ABB RAPID module: 0017732A

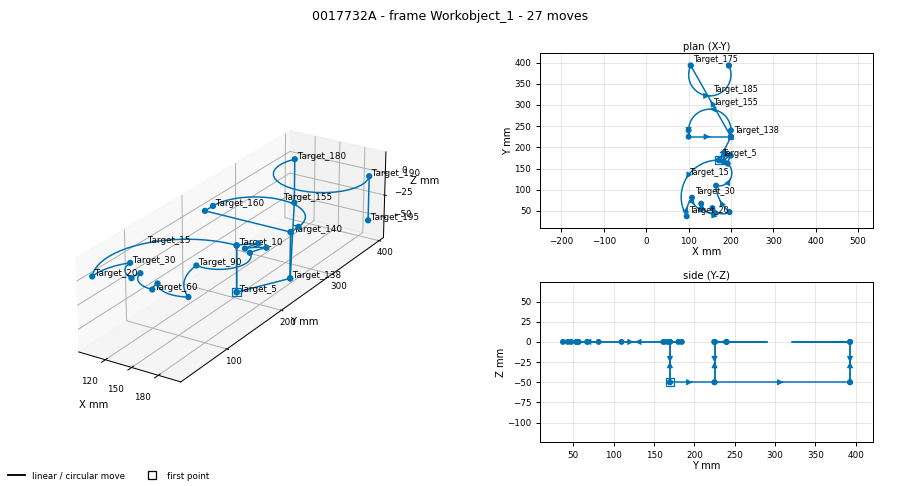
[picture p0: tool path of 0017732A in frame Workobject_1, 27 of 30 moves have a stored position in this frame; points joined in program order, loops and branches not executed]
MODULE Module1
    CONST robtarget Target_M:=[[-410.514648889,1245.713795009,-649.374024814],[0.613768807,0.08026289,-0.406843498,-0.671806585],[0,-1,0,0],[9E+09,9E+09,9E+09,9E+09,9E+09,9E+09]];
    CONST robtarget Target_HH:=[[580.651275023,0,538.588646413],[0.130526193,0,0.991444861,0],[0,0,0,0],[9E+09,9E+09,9E+09,9E+09,9E+09,9E+09]];
    CONST robtarget Target_5:=[[172.146,169.721,-50],[0,0,0,1],[0,0,-1,1],[9E+09,9E+09,9E+09,9E+09,9E+09,9E+09]];
    CONST robtarget Target_10:=[[172.146,169.721,0],[0,0,0,1],[0,0,-1,1],[9E+09,9E+09,9E+09,9E+09,9E+09,9E+09]];
    CONST robtarget Target_15:=[[94.179,126.363,0],[0,0,0,1],[0,0,-1,1],[9E+09,9E+09,9E+09,9E+09,9E+09,9E+09]];
    CONST robtarget Target_20:=[[95.464,37.16,0],[0,0,0,1],[0,0,-1,1],[9E+09,9E+09,9E+09,9E+09,9E+09,9E+09]];
    CONST robtarget Target_25:=[[97.319,60.55,0],[0,0,0,1],[0,0,-1,1],[9E+09,9E+09,9E+09,9E+09,9E+09,9E+09]];
    CONST robtarget Target_30:=[[108.141,81.369,0],[0,0,0,1],[0,0,-1,1],[9E+09,9E+09,9E+09,9E+09,9E+09,9E+09]];
    CONST robtarget Target_35:=[[114.101,64.13,0],[0,0,0,1],[0,0,-1,1],[9E+09,9E+09,9E+09,9E+09,9E+09,9E+09]];
    CONST robtarget Target_40:=[[128.91,53.479,0],[0,0,0,1],[0,0,-1,1],[9E+09,9E+09,9E+09,9E+09,9E+09,9E+09]];
    CONST robtarget Target_45:=[[128.569,60.297,0],[0,0,0,1],[0,0,-1,1],[9E+09,9E+09,9E+09,9E+09,9E+09,9E+09]];
    CONST robtarget Target_50:=[[129.686,67.033,0],[0,0,0,1],[0,0,-1,1],[9E+09,9E+09,9E+09,9E+09,9E+09,9E+09]];
    CONST robtarget Target_55:=[[140.077,49.513,0],[0,0,0,1],[0,0,-1,1],[9E+09,9E+09,9E+09,9E+09,9E+09,9E+09]];
    CONST robtarget Target_60:=[[159.408,43.089,0],[0,0,0,1],[0,0,-1,1],[9E+09,9E+09,9E+09,9E+09,9E+09,9E+09]];
    CONST robtarget Target_65:=[[156.802,49.64,0],[0,0,0,1],[0,0,-1,1],[9E+09,9E+09,9E+09,9E+09,9E+09,9E+09]];
    CONST robtarget Target_70:=[[156.139,56.659,0],[0,0,0,1],[0,0,-1,1],[9E+09,9E+09,9E+09,9E+09,9E+09,9E+09]];
    CONST robtarget Target_75:=[[174.493,43.802,0],[0,0,0,1],[0,0,-1,1],[9E+09,9E+09,9E+09,9E+09,9E+09,9E+09]];
    CONST robtarget Target_80:=[[196.643,47.198,0],[0,0,0,1],[0,0,-1,1],[9E+09,9E+09,9E+09,9E+09,9E+09,9E+09]];
    CONST robtarget Target_85:=[[173.907,75.001,0],[0,0,0,1],[0,0,-1,1],[9E+09,9E+09,9E+09,9E+09,9E+09,9E+09]];
    CONST robtarget Target_90:=[[164.745,109.728,0],[0,0,0,1],[0,0,-1,1],[9E+09,9E+09,9E+09,9E+09,9E+09,9E+09]];
    CONST robtarget Target_95:=[[198.416,125.037,0],[0,0,0,1],[0,0,-1,1],[9E+09,9E+09,9E+09,9E+09,9E+09,9E+09]];
    CONST robtarget Target_100:=[[192.364,161.526,0],[0,0,0,1],[0,0,-1,1],[9E+09,9E+09,9E+09,9E+09,9E+09,9E+09]];
    CONST robtarget Target_105:=[[195.069,171.202,0],[0,0,0,1],[0,0,-1,1],[9E+09,9E+09,9E+09,9E+09,9E+09,9E+09]];
    CONST robtarget Target_110:=[[199.539,180.201,0],[0,0,0,1],[0,0,-1,1],[9E+09,9E+09,9E+09,9E+09,9E+09,9E+09]];
    CONST robtarget Target_115:=[[190.171,175.306,0],[0,0,0,1],[0,0,-1,1],[9E+09,9E+09,9E+09,9E+09,9E+09,9E+09]];
    CONST robtarget Target_120:=[[183.068,167.479,0],[0,0,0,1],[0,0,-1,1],[9E+09,9E+09,9E+09,9E+09,9E+09,9E+09]];
    CONST robtarget Target_125:=[[184.555,176.204,0],[0,0,0,1],[0,0,-1,1],[9E+09,9E+09,9E+09,9E+09,9E+09,9E+09]];
    CONST robtarget Target_130:=[[187.549,184.533,0],[0,0,0,1],[0,0,-1,1],[9E+09,9E+09,9E+09,9E+09,9E+09,9E+09]];
    CONST robtarget Target_135:=[[179.202,177.798,0],[0,0,0,1],[0,0,-1,1],[9E+09,9E+09,9E+09,9E+09,9E+09,9E+09]];
    CONST robtarget Target_138:=[[200,225,-50],[0,0,0,1],[0,-1,0,1],[9E+09,9E+09,9E+09,9E+09,9E+09,9E+09]];
    CONST robtarget Target_140:=[[200,225,0],[0,0,0,1],[0,-1,0,1],[9E+09,9E+09,9E+09,9E+09,9E+09,9E+09]];
    CONST robtarget Target_150:=[[200,240,0],[0,0,0,1],[-1,-1,0,1],[9E+09,9E+09,9E+09,9E+09,9E+09,9E+09]];
    CONST robtarget Target_155:=[[150,290,0],[0,0,0,1],[-1,-1,0,1],[9E+09,9E+09,9E+09,9E+09,9E+09,9E+09]];
    CONST robtarget Target_160:=[[100,240,0],[0,0,0,1],[-1,-1,0,1],[9E+09,9E+09,9E+09,9E+09,9E+09,9E+09]];
    CONST robtarget Target_170:=[[100,225,0],[0,0,0,1],[0,-1,0,1],[9E+09,9E+09,9E+09,9E+09,9E+09,9E+09]];
    CONST robtarget Target_175:=[[105,392.992,-50],[0,0,0,1],[-1,-1,0,1],[9E+09,9E+09,9E+09,9E+09,9E+09,9E+09]];
    CONST robtarget Target_180:=[[105,392.992,0],[0,0,0,1],[-1,-1,0,1],[9E+09,9E+09,9E+09,9E+09,9E+09,9E+09]];
    CONST robtarget Target_185:=[[150,321.197,0],[0,0,0,1],[-1,-1,0,1],[9E+09,9E+09,9E+09,9E+09,9E+09,9E+09]];
    CONST robtarget Target_190:=[[195,392.992,0],[0,0,0,1],[-1,-1,0,1],[9E+09,9E+09,9E+09,9E+09,9E+09,9E+09]];
    CONST robtarget Target_195:=[[195,392.992,-50],[0,0,0,1],[-1,-1,0,1],[9E+09,9E+09,9E+09,9E+09,9E+09,9E+09]];
    CONST robtarget Target_H:=[[-350,1055.651275023,-538.588646413],[0.701057385,-0.092295956,-0.092295956,-0.701057385],[0,0,0,0],[9E+09,9E+09,9E+09,9E+09,9E+09,9E+09]];
    CONST robtarget Target_MM:=[[770.713816879,-60.514661016,649.373982496],[0.230927375,-0.041038912,0.909039083,-0.344436207],[0,-1,0,0],[9E+09,9E+09,9E+09,9E+09,9E+09,9E+09]];
    PROC main()
        Reset DO_01;
        Reset DO_02;
        WHILE TRUE DO
            IF DI_01=1 THEN
                Set DO_01;
                Twitter;
                Reset DO_01;
            ENDIF
            IF DI_02=1 THEN
                Set DO_02;
                Path_40;
                Reset DO_02;
            ENDIF
        ENDWHILE
    ENDPROC
    PROC Path_40()
        MoveJ Target_MM,v600,z0,THerramienta\WObj:=wobj0;
    ENDPROC
    PROC Twitter()
        MoveJ Target_HH,v600,z0,THerramienta\WObj:=wobj0;
        MoveJ Target_5,v600,z5,THerramienta\WObj:=Workobject_1;
        MoveL Target_10,v200,z0,THerramienta\WObj:=Workobject_1;
        MoveC Target_15,Target_20,v200,z0,THerramienta\WObj:=Workobject_1;
        MoveC Target_25,Target_30,v200,z0,THerramienta\WObj:=Workobject_1;
        MoveC Target_35,Target_40,v200,z0,THerramienta\WObj:=Workobject_1;
        MoveC Target_45,Target_50,v200,z0,THerramienta\WObj:=Workobject_1;
        MoveC Target_55,Target_60,v200,z0,THerramienta\WObj:=Workobject_1;
        MoveC Target_65,Target_70,v200,z0,THerramienta\WObj:=Workobject_1;
        MoveC Target_75,Target_80,v200,z0,THerramienta\WObj:=Workobject_1;
        MoveC Target_85,Target_90,v200,z0,THerramienta\WObj:=Workobject_1;
        MoveC Target_95,Target_100,v200,z0,THerramienta\WObj:=Workobject_1;
        MoveC Target_105,Target_110,v200,z0,THerramienta\WObj:=Workobject_1;
        MoveC Target_115,Target_120,v200,z0,THerramienta\WObj:=Workobject_1;
        MoveC Target_125,Target_130,v200,z0,THerramienta\WObj:=Workobject_1;
        MoveC Target_135,Target_10,v200,z0,THerramienta\WObj:=Workobject_1;
        MoveL Target_5,v200,z0,THerramienta\WObj:=Workobject_1;
        MoveL Target_138,v200,z0,THerramienta\WObj:=Workobject_1;
        MoveL Target_140,v200,z0,THerramienta\WObj:=Workobject_1;
        MoveL Target_150,v200,z0,THerramienta\WObj:=Workobject_1;
        MoveC Target_155,Target_160,v200,z0,THerramienta\WObj:=Workobject_1;
        MoveL Target_170,v200,z0,THerramienta\WObj:=Workobject_1;
        MoveL Target_140,v200,z0,THerramienta\WObj:=Workobject_1;
        MoveL Target_138,v200,z0,THerramienta\WObj:=Workobject_1;
        MoveL Target_175,v200,z0,THerramienta\WObj:=Workobject_1;
        MoveL Target_180,v200,z0,THerramienta\WObj:=Workobject_1;
        MoveC Target_185,Target_190,v200,z0,THerramienta\WObj:=Workobject_1;
        MoveL Target_195,v200,z0,THerramienta\WObj:=Workobject_1;
        MoveJ Target_HH,v600,z0,THerramienta\WObj:=wobj0;
    ENDPROC
ENDMODULE
